// TIA Portal V20 export
// export: Created 2026-04-11T06:02:30.5164654Z, ExportSetting WithDefaults, DisplayName Totally Integrated Automation Portal, DisplayVersion V20, DisplayName TIA Portal Openness, DisplayVersion V20, DisplayName TIA Portal Version Control Interface, DisplayVersion V20, DisplayName STEP 7 Professional, DisplayVersion V20, DisplayName STEP 7 Safety, DisplayVersion V20, DisplayName WinCC Basic/Comfort/Advanced, DisplayVersion V20, DisplayName WinCC Unified, DisplayVersion V20
TYPE "udtHMI_HopperControl_Status"
// stored: IsFailsafeCompliant false
   STRUCT
      bError { ExternalWritable := 'False'} : Bool;   // General error
      bLLProcess { ExternalWritable := 'False'} : Bool;   // Bulk Tank Low Level
      bHLProcess { ExternalWritable := 'False'} : Bool;   // Bulk Tank High Level
      bLLAlarm { ExternalWritable := 'False'} : Bool;   // High level alarm
      bHLAlarm { ExternalWritable := 'False'} : Bool;   // Low level alarm
      rLevel { ExternalWritable := 'False'} : Real;   // Actual level
      iStatus { ExternalWritable := 'False'} : Int;   // Status value
   END_STRUCT;
END_TYPE
